(* IEC 61131-3 sources: mocks/test, 17 files *)

(* ---- dummytest.st ---- *)
NAMESPACE dummy
    {Test}
    FUNCTION MyTest
      ; // AxUnit.Assert.Equal(y, x)
    END_FUNCTION
END_NAMESPACE

(* ---- ConfigurableTimerMockTest.st ---- *)
USING System.Timer;
USING AxUnit.Assert;

NAMESPACE Simatic.Ax.Mocks
    /// Example function block that uses multiple OnDelay timers
    FUNCTION_BLOCK MultiTimerFunctionBlock
        VAR_INPUT
            enable1 : BOOL;
            enable2 : BOOL;
            enable3 : BOOL;
        END_VAR
        VAR_OUTPUT
            status1 : STRING;
            status2 : STRING;
            status3 : STRING;
        END_VAR
        VAR
            timer1 : OnDelay;
            timer2 : OnDelay;
            timer3 : OnDelay;
        END_VAR

        // Timer 1: 1 second delay
        timer1(signal := enable1, duration := T#1s);
        IF timer1.output THEN
            status1 := 'T1_ELAPSED';
        ELSE
            status1 := 'T1_WAITING';
        END_IF;

        // Timer 2: 2 second delay
        timer2(signal := enable2, duration := T#2s);
        IF timer2.output THEN
            status2 := 'T2_ELAPSED';
        ELSE
            status2 := 'T2_WAITING';
        END_IF;

        // Timer 3: 5 second delay
        timer3(signal := enable3, duration := T#5s);
        IF timer3.output THEN
            status3 := 'T3_ELAPSED';
        ELSE
            status3 := 'T3_WAITING';
        END_IF;
    END_FUNCTION_BLOCK

    /// Test fixture demonstrating ConfigurableTimerMock usage
    {TestFixture}
    CLASS TestConfigurableTimerMock
        VAR
            testInstance, testInstanceStateless : MultiTimerFunctionBlock;
            payload, payloadStateless : ConfigurableTimerMockPayload;
        END_VAR

        /// Setup method to reset instances before each test
        {TestSetup}
        METHOD PUBLIC TestSetup
            payload := payloadStateless;
            testInstance := testInstanceStateless;
        END_METHOD

        /// Test with Timer 1 elapsed, Timer 2 waiting, Timer 3 elapsed
        /// Timers are identified by call order: 1st call = T1, 2nd call = T2, 3rd call = T3
        {Test}
        METHOD PUBLIC TestMultipleTimersWithDifferentStates
            // Reset counter before test
            payload.ResetCounter();

            // Configure payload: T1=TRUE, T2=FALSE, T3=TRUE (by call order)
            payload.T1_Enabled := TRUE;
            payload.T1_Output := TRUE;
            payload.T1_ElapsedTime := T#1s;

            payload.T2_Enabled := TRUE;
            payload.T2_Output := FALSE;
            payload.T2_ElapsedTime := T#500ms;

            payload.T3_Enabled := TRUE;
            payload.T3_Output := TRUE;
            payload.T3_ElapsedTime := T#5s;

            // Apply mock with payload
            AxUnit.Mocking.Mock(
                mockeeFn := NAME_OF(OnDelay),
                mockFn := NAME_OF(ConfigurableTimerMock),
                payload := payload
            );

            // Execute function block
            // Timer calls happen in order: timer1 (1st call), timer2 (2nd call), timer3 (3rd call)
            testInstance(enable1 := TRUE, enable2 := TRUE, enable3 := TRUE);

            // Verify results
            Equal(expected := 'T1_ELAPSED', actual := testInstance.status1);
            Equal(expected := 'T2_WAITING', actual := testInstance.status2);
            Equal(expected := 'T3_ELAPSED', actual := testInstance.status3);
        END_METHOD

        /// Test with all timers elapsed
        {Test}
        METHOD PUBLIC TestAllTimersElapsed
            // Reset counter before test
            payload.ResetCounter();

            // Configure payload: All timers elapsed
            payload.T1_Enabled := TRUE;
            payload.T1_Output := TRUE;
            payload.T1_ElapsedTime := T#1s;

            payload.T2_Enabled := TRUE;
            payload.T2_Output := TRUE;
            payload.T2_ElapsedTime := T#2s;

            payload.T3_Enabled := TRUE;
            payload.T3_Output := TRUE;
            payload.T3_ElapsedTime := T#5s;

            // Apply mock with payload
            AxUnit.Mocking.Mock(
                mockeeFn := NAME_OF(OnDelay),
                mockFn := NAME_OF(ConfigurableTimerMock),
                payload := payload
            );

            // Execute function block
            testInstance(enable1 := TRUE, enable2 := TRUE, enable3 := TRUE);

            // Verify results
            Equal(expected := 'T1_ELAPSED', actual := testInstance.status1);
            Equal(expected := 'T2_ELAPSED', actual := testInstance.status2);
            Equal(expected := 'T3_ELAPSED', actual := testInstance.status3);
        END_METHOD

        /// Test with only Timer 2 enabled (2nd call)
        {Test}
        METHOD PUBLIC TestOnlyTimer2Enabled
            // Reset counter before test
            payload.ResetCounter();

            // Configure payload: Only T2 enabled and elapsed
            payload.T1_Enabled := FALSE;  // 1st call returns FALSE

            payload.T2_Enabled := TRUE;   // 2nd call returns TRUE
            payload.T2_Output := TRUE;
            payload.T2_ElapsedTime := T#2s;

            payload.T3_Enabled := FALSE;  // 3rd call returns FALSE

            // Apply mock with payload
            AxUnit.Mocking.Mock(
                mockeeFn := NAME_OF(OnDelay),
                mockFn := NAME_OF(ConfigurableTimerMock),
                payload := payload
            );

            // Execute function block
            testInstance(enable1 := TRUE, enable2 := TRUE, enable3 := TRUE);

            // Verify results
            Equal(expected := 'T1_WAITING', actual := testInstance.status1); // 1st call: not enabled
            Equal(expected := 'T2_ELAPSED', actual := testInstance.status2); // 2nd call: enabled and TRUE
            Equal(expected := 'T3_WAITING', actual := testInstance.status3); // 3rd call: not enabled
        END_METHOD
    END_CLASS
END_NAMESPACE

(* ---- ConfigurableTOFMockTest.st ---- *)
USING AxUnit.Assert;

NAMESPACE Simatic.Ax.Mocks
    /// Example function block that uses multiple TOF timers
    FUNCTION_BLOCK MultiTOFFunctionBlock
        VAR_INPUT
            enable1 : BOOL;
            enable2 : BOOL;
            enable3 : BOOL;
        END_VAR
        VAR_OUTPUT
            status1 : STRING;
            status2 : STRING;
            status3 : STRING;
        END_VAR
        VAR
            timer1 : TOF_Mock_true;
            timer2 : TOF_Mock_true;
            timer3 : TOF_Mock_true;
        END_VAR

        // Timer 1: 1 second delay
        timer1(IN := enable1, PT := T#1s);
        IF timer1.Q THEN
            status1 := 'T1_ON';
        ELSE
            status1 := 'T1_OFF';
        END_IF;

        // Timer 2: 2 second delay
        timer2(IN := enable2, PT := T#2s);
        IF timer2.Q THEN
            status2 := 'T2_ON';
        ELSE
            status2 := 'T2_OFF';
        END_IF;

        // Timer 3: 5 second delay
        timer3(IN := enable3, PT := T#5s);
        IF timer3.Q THEN
            status3 := 'T3_ON';
        ELSE
            status3 := 'T3_OFF';
        END_IF;
    END_FUNCTION_BLOCK

    /// Test fixture demonstrating ConfigurableTOFMock usage
    {TestFixture}
    CLASS TestConfigurableTOFMock
        VAR
            testInstance, testInstanceStateless : MultiTOFFunctionBlock;
            payload, payloadStateless : ConfigurableTOFMockPayload;
        END_VAR

        /// Setup method to reset instances before each test
        {TestSetup}
        METHOD PUBLIC TestSetup
            payload := payloadStateless;
            testInstance := testInstanceStateless;
        END_METHOD

        /// Test with Timer 1 ON, Timer 2 OFF, Timer 3 ON
        /// Timers are identified by call order: 1st call = T1, 2nd call = T2, 3rd call = T3
        {Test}
        METHOD PUBLIC TestMultipleTimersWithDifferentStates
            // Reset counter before test
            payload.ResetCounter();

            // Configure payload: T1=TRUE, T2=FALSE, T3=TRUE (by call order)
            payload.T1_Enabled := TRUE;
            payload.T1_Output := TRUE;
            payload.T1_ElapsedTime := T#0ms;

            payload.T2_Enabled := TRUE;
            payload.T2_Output := FALSE;
            payload.T2_ElapsedTime := T#2s;

            payload.T3_Enabled := TRUE;
            payload.T3_Output := TRUE;
            payload.T3_ElapsedTime := T#0ms;

            // Apply mock with payload
            AxUnit.Mocking.Mock(
                mockeeFn := NAME_OF(TOF_Mock_true),
                mockFn := NAME_OF(ConfigurableTOFMock),
                payload := payload
            );

            // Execute function block
            // Timer calls happen in order: timer1 (1st call), timer2 (2nd call), timer3 (3rd call)
            testInstance(enable1 := FALSE, enable2 := FALSE, enable3 := FALSE);

            // Verify results
            Equal(expected := 'T1_ON', actual := testInstance.status1);
            Equal(expected := 'T2_OFF', actual := testInstance.status2);
            Equal(expected := 'T3_ON', actual := testInstance.status3);
        END_METHOD

        /// Test with all timers OFF (delay elapsed)
        {Test}
        METHOD PUBLIC TestAllTimersOff
            // Reset counter before test
            payload.ResetCounter();

            // Configure payload: All timers OFF
            payload.T1_Enabled := TRUE;
            payload.T1_Output := FALSE;
            payload.T1_ElapsedTime := T#1s;

            payload.T2_Enabled := TRUE;
            payload.T2_Output := FALSE;
            payload.T2_ElapsedTime := T#2s;

            payload.T3_Enabled := TRUE;
            payload.T3_Output := FALSE;
            payload.T3_ElapsedTime := T#5s;

            // Apply mock with payload
            AxUnit.Mocking.Mock(
                mockeeFn := NAME_OF(TOF_Mock_true),
                mockFn := NAME_OF(ConfigurableTOFMock),
                payload := payload
            );

            // Execute function block
            testInstance(enable1 := FALSE, enable2 := FALSE, enable3 := FALSE);

            // Verify results
            Equal(expected := 'T1_OFF', actual := testInstance.status1);
            Equal(expected := 'T2_OFF', actual := testInstance.status2);
            Equal(expected := 'T3_OFF', actual := testInstance.status3);
        END_METHOD

        /// Test with only Timer 2 enabled (2nd call)
        {Test}
        METHOD PUBLIC TestOnlyTimer2Enabled
            // Reset counter before test
            payload.ResetCounter();

            // Configure payload: Only T2 enabled and ON
            payload.T1_Enabled := FALSE;  // 1st call returns FALSE

            payload.T2_Enabled := TRUE;   // 2nd call returns TRUE
            payload.T2_Output := TRUE;
            payload.T2_ElapsedTime := T#0ms;

            payload.T3_Enabled := FALSE;  // 3rd call returns FALSE

            // Apply mock with payload
            AxUnit.Mocking.Mock(
                mockeeFn := NAME_OF(TOF_Mock_true),
                mockFn := NAME_OF(ConfigurableTOFMock),
                payload := payload
            );

            // Execute function block
            testInstance(enable1 := FALSE, enable2 := FALSE, enable3 := FALSE);

            // Verify results
            Equal(expected := 'T1_OFF', actual := testInstance.status1); // 1st call: not enabled
            Equal(expected := 'T2_ON', actual := testInstance.status2);  // 2nd call: enabled and TRUE
            Equal(expected := 'T3_OFF', actual := testInstance.status3); // 3rd call: not enabled
        END_METHOD

        /// Test with all timers ON (signal still active or delay not elapsed)
        {Test}
        METHOD PUBLIC TestAllTimersOn
            // Reset counter before test
            payload.ResetCounter();

            // Configure payload: All timers ON
            payload.T1_Enabled := TRUE;
            payload.T1_Output := TRUE;
            payload.T1_ElapsedTime := T#0ms;

            payload.T2_Enabled := TRUE;
            payload.T2_Output := TRUE;
            payload.T2_ElapsedTime := T#0ms;

            payload.T3_Enabled := TRUE;
            payload.T3_Output := TRUE;
            payload.T3_ElapsedTime := T#0ms;

            // Apply mock with payload
            AxUnit.Mocking.Mock(
                mockeeFn := NAME_OF(TOF_Mock_true),
                mockFn := NAME_OF(ConfigurableTOFMock),
                payload := payload
            );

            // Execute function block
            testInstance(enable1 := TRUE, enable2 := TRUE, enable3 := TRUE);

            // Verify results
            Equal(expected := 'T1_ON', actual := testInstance.status1);
            Equal(expected := 'T2_ON', actual := testInstance.status2);
            Equal(expected := 'T3_ON', actual := testInstance.status3);
        END_METHOD
    END_CLASS
END_NAMESPACE

(* ---- ConfigurableTONMockTest.st ---- *)
USING AxUnit.Assert;

NAMESPACE Simatic.Ax.Mocks
    /// Example function block that uses multiple TON timers
    FUNCTION_BLOCK MultiTONFunctionBlock
        VAR_INPUT
            enable1 : BOOL;
            enable2 : BOOL;
            enable3 : BOOL;
        END_VAR
        VAR_OUTPUT
            status1 : STRING;
            status2 : STRING;
            status3 : STRING;
        END_VAR
        VAR
            timer1 : TON_Mock_true;
            timer2 : TON_Mock_true;
            timer3 : TON_Mock_true;
        END_VAR

        // Timer 1: 1 second delay
        timer1(IN := enable1, PT := T#1s);
        IF timer1.Q THEN
            status1 := 'T1_ELAPSED';
        ELSE
            status1 := 'T1_WAITING';
        END_IF;

        // Timer 2: 2 second delay
        timer2(IN := enable2, PT := T#2s);
        IF timer2.Q THEN
            status2 := 'T2_ELAPSED';
        ELSE
            status2 := 'T2_WAITING';
        END_IF;

        // Timer 3: 5 second delay
        timer3(IN := enable3, PT := T#5s);
        IF timer3.Q THEN
            status3 := 'T3_ELAPSED';
        ELSE
            status3 := 'T3_WAITING';
        END_IF;
    END_FUNCTION_BLOCK

    /// Test fixture demonstrating ConfigurableTONMock usage
    {TestFixture}
    CLASS TestConfigurableTONMock
        VAR
            testInstance, testInstanceStateless : MultiTONFunctionBlock;
            payload, payloadStateless : ConfigurableTONMockPayload;
        END_VAR

        /// Setup method to reset instances before each test
        {TestSetup}
        METHOD PUBLIC TestSetup
            payload := payloadStateless;
            testInstance := testInstanceStateless;
        END_METHOD

        /// Test with Timer 1 elapsed, Timer 2 waiting, Timer 3 elapsed
        /// Timers are identified by call order: 1st call = T1, 2nd call = T2, 3rd call = T3
        {Test}
        METHOD PUBLIC TestMultipleTimersWithDifferentStates
            // Reset counter before test
            payload.ResetCounter();

            // Configure payload: T1=TRUE, T2=FALSE, T3=TRUE (by call order)
            payload.T1_Enabled := TRUE;
            payload.T1_Output := TRUE;
            payload.T1_ElapsedTime := T#1s;

            payload.T2_Enabled := TRUE;
            payload.T2_Output := FALSE;
            payload.T2_ElapsedTime := T#500ms;

            payload.T3_Enabled := TRUE;
            payload.T3_Output := TRUE;
            payload.T3_ElapsedTime := T#5s;

            // Apply mock with payload
            AxUnit.Mocking.Mock(
                mockeeFn := NAME_OF(TON_Mock_true),
                mockFn := NAME_OF(ConfigurableTONMock),
                payload := payload
            );

            // Execute function block
            // Timer calls happen in order: timer1 (1st call), timer2 (2nd call), timer3 (3rd call)
            testInstance(enable1 := TRUE, enable2 := TRUE, enable3 := TRUE);

            // Verify results
            Equal(expected := 'T1_ELAPSED', actual := testInstance.status1);
            Equal(expected := 'T2_WAITING', actual := testInstance.status2);
            Equal(expected := 'T3_ELAPSED', actual := testInstance.status3);
        END_METHOD

        /// Test with all timers elapsed
        {Test}
        METHOD PUBLIC TestAllTimersElapsed
            // Reset counter before test
            payload.ResetCounter();

            // Configure payload: All timers elapsed
            payload.T1_Enabled := TRUE;
            payload.T1_Output := TRUE;
            payload.T1_ElapsedTime := T#1s;

            payload.T2_Enabled := TRUE;
            payload.T2_Output := TRUE;
            payload.T2_ElapsedTime := T#2s;

            payload.T3_Enabled := TRUE;
            payload.T3_Output := TRUE;
            payload.T3_ElapsedTime := T#5s;

            // Apply mock with payload
            AxUnit.Mocking.Mock(
                mockeeFn := NAME_OF(TON_Mock_true),
                mockFn := NAME_OF(ConfigurableTONMock),
                payload := payload
            );

            // Execute function block
            testInstance(enable1 := TRUE, enable2 := TRUE, enable3 := TRUE);

            // Verify results
            Equal(expected := 'T1_ELAPSED', actual := testInstance.status1);
            Equal(expected := 'T2_ELAPSED', actual := testInstance.status2);
            Equal(expected := 'T3_ELAPSED', actual := testInstance.status3);
        END_METHOD

        /// Test with only Timer 2 enabled (2nd call)
        {Test}
        METHOD PUBLIC TestOnlyTimer2Enabled
            // Reset counter before test
            payload.ResetCounter();

            // Configure payload: Only T2 enabled and elapsed
            payload.T1_Enabled := FALSE;  // 1st call returns FALSE

            payload.T2_Enabled := TRUE;   // 2nd call returns TRUE
            payload.T2_Output := TRUE;
            payload.T2_ElapsedTime := T#2s;

            payload.T3_Enabled := FALSE;  // 3rd call returns FALSE

            // Apply mock with payload
            AxUnit.Mocking.Mock(
                mockeeFn := NAME_OF(TON_Mock_true),
                mockFn := NAME_OF(ConfigurableTONMock),
                payload := payload
            );

            // Execute function block
            testInstance(enable1 := TRUE, enable2 := TRUE, enable3 := TRUE);

            // Verify results
            Equal(expected := 'T1_WAITING', actual := testInstance.status1); // 1st call: not enabled
            Equal(expected := 'T2_ELAPSED', actual := testInstance.status2); // 2nd call: enabled and TRUE
            Equal(expected := 'T3_WAITING', actual := testInstance.status3); // 3rd call: not enabled
        END_METHOD

        /// Test with all timers waiting
        {Test}
        METHOD PUBLIC TestAllTimersWaiting
            // Reset counter before test
            payload.ResetCounter();

            // Configure payload: All timers waiting
            payload.T1_Enabled := TRUE;
            payload.T1_Output := FALSE;
            payload.T1_ElapsedTime := T#500ms;

            payload.T2_Enabled := TRUE;
            payload.T2_Output := FALSE;
            payload.T2_ElapsedTime := T#1s;

            payload.T3_Enabled := TRUE;
            payload.T3_Output := FALSE;
            payload.T3_ElapsedTime := T#3s;

            // Apply mock with payload
            AxUnit.Mocking.Mock(
                mockeeFn := NAME_OF(TON_Mock_true),
                mockFn := NAME_OF(ConfigurableTONMock),
                payload := payload
            );

            // Execute function block
            testInstance(enable1 := TRUE, enable2 := TRUE, enable3 := TRUE);

            // Verify results
            Equal(expected := 'T1_WAITING', actual := testInstance.status1);
            Equal(expected := 'T2_WAITING', actual := testInstance.status2);
            Equal(expected := 'T3_WAITING', actual := testInstance.status3);
        END_METHOD
    END_CLASS
END_NAMESPACE

(* ---- ExampleMockTimer.st ---- *)
USING System.Timer;
USING AxUnit.Assert;

NAMESPACE Simatic.Ax.Mocks
    FUNCTION_BLOCK FunctionBlockWhichUsesTimer
        VAR_INPUT
            enable : BOOL;
        END_VAR
        VAR_OUTPUT
            timerStatus : STRING;
        END_VAR

        VAR
            ton : OnDelay;
        END_VAR

        ton(signal := enable, duration := T#10s);

        IF (ton.output) THEN
            timerStatus := 'ELAPSED';
        ELSIF (ton.signal AND NOT ton.output) THEN
            timerStatus := 'RUNNING';
        ELSIF (NOT ton.signal) THEN
            timerStatus := 'IDLE';
        END_IF;
        ;
    END_FUNCTION_BLOCK

    {TestFixture}
    CLASS TestFunctionBlockWhichUsesTimer
        VAR
            testInstance : FunctionBlockWhichUsesTimer;
        END_VAR

        {Test}
        METHOD PUBLIC FunctionBlockReturnsIdleWhenNotEnabled
            testInstance(enable := FALSE);
            Equal(expected := 'ELAPSED', actual := testInstance.timerStatus);
        END_METHOD

        {Test}
        METHOD PUBLIC FunctionBlockReturnsRunningWhenEnabledAndTimeIsNotElapsed
            testInstance(enable := TRUE);
            Equal(expected := 'RUNNING', actual := testInstance.timerStatus);
        END_METHOD

        {Test}
        METHOD PUBLIC FunctionBlockReturnsElapsedWhenEnabledAndTimeHasElapsed
            testInstance(enable := TRUE);
            Equal(expected := 'ELAPSED', actual := testInstance.timerStatus);
        END_METHOD
    END_CLASS
END_NAMESPACE

(* ---- FooFB_ConfigurableMock_Test.st ---- *)
USING AxUnit.Assert;
USING System.Timer;

NAMESPACE Simatic.Ax.Mocks
    /// Test fixture for FbWithThreeTimers using ConfigurableTimerMock
    /// This demonstrates call-order based timer mocking
    /// Uses stateless pattern to ensure test isolation
    {TestFixture}
    CLASS TestFbWithThreeTimers_ConfigurableMock
        VAR
            myFB, myFBStateless : FbWithThreeTimers;
            payload, payloadStateless : ConfigurableTimerMockPayload;
        END_VAR

        /// Setup method to reset instances before each test
        {TestSetup}
        METHOD PUBLIC TestSetup
            payload := payloadStateless;
            myFB := myFBStateless;
        END_METHOD

        /// Test scenario: T1 elapsed, T2 waiting, T3 elapsed
        {Test}
        METHOD PUBLIC Test_T1_Elapsed_T2_Waiting_T3_Elapsed
            // Reset counter before test
            payload.ResetCounter();

            // Configure timers by call order
            // T1 is 1st call - elapsed
            payload.T1_Enabled := TRUE;
            payload.T1_Output := TRUE;
            payload.T1_ElapsedTime := T#10s;

            // T2 is 2nd call - waiting
            payload.T2_Enabled := TRUE;
            payload.T2_Output := FALSE;
            payload.T2_ElapsedTime := T#5s;

            // T3 is 3rd call - elapsed
            payload.T3_Enabled := TRUE;
            payload.T3_Output := TRUE;
            payload.T3_ElapsedTime := T#30s;

            // Apply mock
            AxUnit.Mocking.Mock(
                mockeeFn := NAME_OF(OnDelay),
                mockFn := NAME_OF(ConfigurableTimerMock),
                payload := payload
            );

            // Execute function block
            myFB.SignalT1 := TRUE;
            myFB.SignalT2 := TRUE;
            myFB.SignalT3 := TRUE;
            myFB();

            // Verify results
            Equal(expected := TRUE, actual := myFB.OutputT1);
            Equal(expected := FALSE, actual := myFB.OutputT2);
            Equal(expected := TRUE, actual := myFB.OutputT3);
        END_METHOD

        /// Test scenario: All timers elapsed
        {Test}
        METHOD PUBLIC Test_AllTimersElapsed
            payload.ResetCounter();

            // All timers elapsed
            payload.T1_Enabled := TRUE;
            payload.T1_Output := TRUE;
            payload.T1_ElapsedTime := T#10s;

            payload.T2_Enabled := TRUE;
            payload.T2_Output := TRUE;
            payload.T2_ElapsedTime := T#20s;

            payload.T3_Enabled := TRUE;
            payload.T3_Output := TRUE;
            payload.T3_ElapsedTime := T#30s;

            // Apply mock
            AxUnit.Mocking.Mock(
                mockeeFn := NAME_OF(OnDelay),
                mockFn := NAME_OF(ConfigurableTimerMock),
                payload := payload
            );

            // Execute
            myFB.SignalT1 := TRUE;
            myFB.SignalT2 := TRUE;
            myFB.SignalT3 := TRUE;
            myFB();

            // Verify all outputs are TRUE
            Equal(expected := TRUE, actual := myFB.OutputT1);
            Equal(expected := TRUE, actual := myFB.OutputT2);
            Equal(expected := TRUE, actual := myFB.OutputT3);
        END_METHOD

        /// Test scenario: All timers waiting
        {Test}
        METHOD PUBLIC Test_AllTimersWaiting
            payload.ResetCounter();

            // All timers waiting
            payload.T1_Enabled := TRUE;
            payload.T1_Output := FALSE;
            payload.T1_ElapsedTime := T#3s;

            payload.T2_Enabled := TRUE;
            payload.T2_Output := FALSE;
            payload.T2_ElapsedTime := T#7s;

            payload.T3_Enabled := TRUE;
            payload.T3_Output := FALSE;
            payload.T3_ElapsedTime := T#15s;

            // Apply mock
            AxUnit.Mocking.Mock(
                mockeeFn := NAME_OF(OnDelay),
                mockFn := NAME_OF(ConfigurableTimerMock),
                payload := payload
            );

            // Execute
            myFB.SignalT1 := TRUE;
            myFB.SignalT2 := TRUE;
            myFB.SignalT3 := TRUE;
            myFB();

            // Verify all outputs are FALSE
            Equal(expected := FALSE, actual := myFB.OutputT1);
            Equal(expected := FALSE, actual := myFB.OutputT2);
            Equal(expected := FALSE, actual := myFB.OutputT3);
        END_METHOD

        /// Test scenario: Only T2 enabled (others disabled)
        {Test}
        METHOD PUBLIC Test_OnlyT2Enabled
            payload.ResetCounter();

            // Only T2 enabled at position 2
            payload.T1_Enabled := FALSE;  // 1st call - not configured

            payload.T2_Enabled := TRUE;   // 2nd call - configured
            payload.T2_Output := TRUE;
            payload.T2_ElapsedTime := T#20s;

            payload.T3_Enabled := FALSE;  // 3rd call - not configured

            // Apply mock
            AxUnit.Mocking.Mock(
                mockeeFn := NAME_OF(OnDelay),
                mockFn := NAME_OF(ConfigurableTimerMock),
                payload := payload
            );

            // Execute
            myFB.SignalT1 := TRUE;
            myFB.SignalT2 := TRUE;
            myFB.SignalT3 := TRUE;
            myFB();

            // Verify: T1 and T3 default to FALSE, T2 is TRUE
            Equal(expected := FALSE, actual := myFB.OutputT1);
            Equal(expected := TRUE, actual := myFB.OutputT2);
            Equal(expected := FALSE, actual := myFB.OutputT3);
        END_METHOD

        /// Test scenario: Mixed signals - some enabled, some disabled
        {Test}
        METHOD PUBLIC Test_MixedSignals
            payload.ResetCounter();

            // Configure all timers as elapsed
            payload.T1_Enabled := TRUE;
            payload.T1_Output := TRUE;
            payload.T1_ElapsedTime := T#10s;

            payload.T2_Enabled := TRUE;
            payload.T2_Output := TRUE;
            payload.T2_ElapsedTime := T#20s;

            payload.T3_Enabled := TRUE;
            payload.T3_Output := TRUE;
            payload.T3_ElapsedTime := T#30s;

            // Apply mock
            AxUnit.Mocking.Mock(
                mockeeFn := NAME_OF(OnDelay),
                mockFn := NAME_OF(ConfigurableTimerMock),
                payload := payload
            );

            // Execute with mixed signals
            myFB.SignalT1 := TRUE;   // Enabled
            myFB.SignalT2 := FALSE;  // Disabled
            myFB.SignalT3 := TRUE;   // Enabled
            myFB();

            // Verify: Mock returns configured values regardless of signal
            // (This is the mock behavior - it ignores the signal input)
            Equal(expected := TRUE, actual := myFB.OutputT1);
            Equal(expected := TRUE, actual := myFB.OutputT2);
            Equal(expected := TRUE, actual := myFB.OutputT3);
        END_METHOD
    END_CLASS
END_NAMESPACE

(* ---- FooFB_IdentifierMock_Test.st ---- *)
USING AxUnit.Assert;
USING System.Timer;

NAMESPACE Simatic.Ax.Mocks
    /// Test fixture for FbWithThreeTimers using IdentifierBasedTimerMock
    /// This demonstrates position-based timer mocking with explicit call positions
    /// Uses stateless pattern to ensure test isolation
    {TestFixture}
    CLASS TestFbWithThreeTimers_IdentifierMock
        VAR
            myFB, myFBStateless : FbWithThreeTimers;
            payload, payloadStateless : IdentifierBasedOnDelayMockPayload;
        END_VAR

        /// Setup method to reset instances before each test
        {TestSetup}
        METHOD PUBLIC TestSetup
            payload := payloadStateless;
            myFB := myFBStateless;
        END_METHOD

        /// Test scenario: T1 elapsed, T2 waiting, T3 elapsed
        /// Using explicit call positions
        {Test}
        METHOD PUBLIC Test_T1_Elapsed_T2_Waiting_T3_Elapsed
            // Reset counter before test
            payload.ResetCounter();

            // Configure timers by explicit call position
            // T1 at position 1 - elapsed
            payload.T1_Enabled := TRUE;
            payload.T1_CallPosition := 1;  // 1st call
            payload.T1_Output := TRUE;
            payload.T1_ElapsedTime := T#10s;

            // T2 at position 2 - waiting
            payload.T2_Enabled := TRUE;
            payload.T2_CallPosition := 2;  // 2nd call
            payload.T2_Output := FALSE;
            payload.T2_ElapsedTime := T#5s;

            // T3 at position 3 - elapsed
            payload.T3_Enabled := TRUE;
            payload.T3_CallPosition := 3;  // 3rd call
            payload.T3_Output := TRUE;
            payload.T3_ElapsedTime := T#30s;

            // Apply mock
            AxUnit.Mocking.Mock(
                mockeeFn := NAME_OF(OnDelay),
                mockFn := NAME_OF(IdentifierBasedOnDelayMock),
                payload := payload
            );

            // Execute function block
            myFB.SignalT1 := TRUE;
            myFB.SignalT2 := TRUE;
            myFB.SignalT3 := TRUE;
            myFB();

            // Verify results
            Equal(expected := TRUE, actual := myFB.OutputT1);
            Equal(expected := FALSE, actual := myFB.OutputT2);
            Equal(expected := TRUE, actual := myFB.OutputT3);
        END_METHOD

        /// Test scenario: All timers elapsed
        {Test}
        METHOD PUBLIC Test_AllTimersElapsed
            payload.ResetCounter();

            // All timers elapsed at their respective positions
            payload.T1_Enabled := TRUE;
            payload.T1_CallPosition := 1;
            payload.T1_Output := TRUE;
            payload.T1_ElapsedTime := T#10s;

            payload.T2_Enabled := TRUE;
            payload.T2_CallPosition := 2;
            payload.T2_Output := TRUE;
            payload.T2_ElapsedTime := T#20s;

            payload.T3_Enabled := TRUE;
            payload.T3_CallPosition := 3;
            payload.T3_Output := TRUE;
            payload.T3_ElapsedTime := T#30s;

            // Apply mock
            AxUnit.Mocking.Mock(
                mockeeFn := NAME_OF(OnDelay),
                mockFn := NAME_OF(IdentifierBasedOnDelayMock),
                payload := payload
            );

            // Execute
            myFB.SignalT1 := TRUE;
            myFB.SignalT2 := TRUE;
            myFB.SignalT3 := TRUE;
            myFB();

            // Verify all outputs are TRUE
            Equal(expected := TRUE, actual := myFB.OutputT1);
            Equal(expected := TRUE, actual := myFB.OutputT2);
            Equal(expected := TRUE, actual := myFB.OutputT3);
        END_METHOD

        /// Test scenario: All timers waiting
        {Test}
        METHOD PUBLIC Test_AllTimersWaiting
            payload.ResetCounter();

            // All timers waiting
            payload.T1_Enabled := TRUE;
            payload.T1_CallPosition := 1;
            payload.T1_Output := FALSE;
            payload.T1_ElapsedTime := T#3s;

            payload.T2_Enabled := TRUE;
            payload.T2_CallPosition := 2;
            payload.T2_Output := FALSE;
            payload.T2_ElapsedTime := T#7s;

            payload.T3_Enabled := TRUE;
            payload.T3_CallPosition := 3;
            payload.T3_Output := FALSE;
            payload.T3_ElapsedTime := T#15s;

            // Apply mock
            AxUnit.Mocking.Mock(
                mockeeFn := NAME_OF(OnDelay),
                mockFn := NAME_OF(IdentifierBasedOnDelayMock),
                payload := payload
            );

            // Execute
            myFB.SignalT1 := TRUE;
            myFB.SignalT2 := TRUE;
            myFB.SignalT3 := TRUE;
            myFB();

            // Verify all outputs are FALSE
            Equal(expected := FALSE, actual := myFB.OutputT1);
            Equal(expected := FALSE, actual := myFB.OutputT2);
            Equal(expected := FALSE, actual := myFB.OutputT3);
        END_METHOD

        /// Test scenario: Only T2 configured at position 2
        {Test}
        METHOD PUBLIC Test_OnlyT2Configured
            payload.ResetCounter();

            // Only configure T2 at position 2
            payload.T1_Enabled := FALSE;  // Position 1 - not configured

            payload.T2_Enabled := TRUE;   // Position 2 - configured
            payload.T2_CallPosition := 2;
            payload.T2_Output := TRUE;
            payload.T2_ElapsedTime := T#20s;

            payload.T3_Enabled := FALSE;  // Position 3 - not configured

            // Apply mock
            AxUnit.Mocking.Mock(
                mockeeFn := NAME_OF(OnDelay),
                mockFn := NAME_OF(IdentifierBasedOnDelayMock),
                payload := payload
            );

            // Execute
            myFB.SignalT1 := TRUE;
            myFB.SignalT2 := TRUE;
            myFB.SignalT3 := TRUE;
            myFB();

            // Verify: T1 and T3 default to FALSE, T2 is TRUE
            Equal(expected := FALSE, actual := myFB.OutputT1);
            Equal(expected := TRUE, actual := myFB.OutputT2);
            Equal(expected := FALSE, actual := myFB.OutputT3);
        END_METHOD

        /// Test scenario: Non-sequential positions (demonstrating flexibility)
        /// Configure T1 at position 3, T3 at position 1 (swapped)
        {Test}
        METHOD PUBLIC Test_NonSequentialPositions
            payload.ResetCounter();

            // Swap positions: T3 at position 1, T1 at position 3
            payload.T1_Enabled := TRUE;
            payload.T1_CallPosition := 3;  // T1 configured for 3rd call
            payload.T1_Output := TRUE;
            payload.T1_ElapsedTime := T#10s;

            payload.T2_Enabled := TRUE;
            payload.T2_CallPosition := 2;  // T2 at 2nd call (normal)
            payload.T2_Output := FALSE;
            payload.T2_ElapsedTime := T#5s;

            payload.T3_Enabled := TRUE;
            payload.T3_CallPosition := 1;  // T3 configured for 1st call
            payload.T3_Output := TRUE;
            payload.T3_ElapsedTime := T#30s;

            // Apply mock
            AxUnit.Mocking.Mock(
                mockeeFn := NAME_OF(OnDelay),
                mockFn := NAME_OF(IdentifierBasedOnDelayMock),
                payload := payload
            );

            // Execute
            myFB.SignalT1 := TRUE;
            myFB.SignalT2 := TRUE;
            myFB.SignalT3 := TRUE;
            myFB();

            // Verify:
            // 1st call (T1 in code) gets T3 config -> TRUE
            // 2nd call (T2 in code) gets T2 config -> FALSE
            // 3rd call (T3 in code) gets T1 config -> TRUE
            Equal(expected := TRUE, actual := myFB.OutputT1);   // Gets T3 config
            Equal(expected := FALSE, actual := myFB.OutputT2);  // Gets T2 config
            Equal(expected := TRUE, actual := myFB.OutputT3);   // Gets T1 config
        END_METHOD

        /// Test scenario: Partial elapsed times
        /// Demonstrates setting specific elapsed times for each timer
        {Test}
        METHOD PUBLIC Test_PartialElapsedTimes
            payload.ResetCounter();

            // Configure with specific elapsed times
            payload.T1_Enabled := TRUE;
            payload.T1_CallPosition := 1;
            payload.T1_Output := FALSE;  // Not elapsed yet
            payload.T1_ElapsedTime := T#7s;  // 7 of 10 seconds

            payload.T2_Enabled := TRUE;
            payload.T2_CallPosition := 2;
            payload.T2_Output := FALSE;  // Not elapsed yet
            payload.T2_ElapsedTime := T#15s;  // 15 of 20 seconds

            payload.T3_Enabled := TRUE;
            payload.T3_CallPosition := 3;
            payload.T3_Output := TRUE;  // Elapsed
            payload.T3_ElapsedTime := T#30s;  // Full 30 seconds

            // Apply mock
            AxUnit.Mocking.Mock(
                mockeeFn := NAME_OF(OnDelay),
                mockFn := NAME_OF(IdentifierBasedOnDelayMock),
                payload := payload
            );

            // Execute
            myFB.SignalT1 := TRUE;
            myFB.SignalT2 := TRUE;
            myFB.SignalT3 := TRUE;
            myFB();

            // Verify outputs
            Equal(expected := FALSE, actual := myFB.OutputT1);  // 7s < 10s
            Equal(expected := FALSE, actual := myFB.OutputT2);  // 15s < 20s
            Equal(expected := TRUE, actual := myFB.OutputT3);   // 30s = 30s
        END_METHOD
    END_CLASS
END_NAMESPACE

(* ---- FooFbWithThreeTimers.st ---- *)
USING AxUnit.Assert;
USING System.Timer;
NAMESPACE Simatic.Ax.Mocks

    FUNCTION_BLOCK FbWithThreeTimers
        VAR_INPUT
            SignalT1 : BOOL;
            SignalT2 : BOOL;
            SignalT3 : BOOL;
        END_VAR
        VAR_OUTPUT
            OutputT1 : BOOL;
            OutputT2 : BOOL;
            OutputT3 : BOOL;
        END_VAR
        VAR
            T1 : OnDelay;
            T2 : OnDelay;
            T3 : OnDelay;
        END_VAR
        T1(Signal := SignalT1, Duration := LTIME#10S, Output => OutputT1);
        T2(Signal := SignalT2, Duration := LTIME#20S, Output => OutputT2);
        T3(Signal := SignalT3, Duration := LTIME#30S, Output => OutputT3);
    END_FUNCTION_BLOCK
END_NAMESPACE

(* ---- IdentifierBasedOffDelayMockTest.st ---- *)
USING System.Timer;
USING AxUnit.Assert;

NAMESPACE Simatic.Ax.Mocks
    /// Example function block with conditional OffDelay timer usage
    FUNCTION_BLOCK ConditionalOffDelayFunctionBlock
        VAR_INPUT
            mode : INT;  // 1, 2, or 3 to select which timer to use
        END_VAR
        VAR_OUTPUT
            result : STRING;
        END_VAR
        VAR
            timer1 : OffDelay;
            timer2 : OffDelay;
            timer3 : OffDelay;
        END_VAR

        // Conditional timer usage based on mode
        IF mode = 1 THEN
            timer1(signal := FALSE, duration := T#1s);
            IF timer1.output THEN
                result := 'MODE1_ON';
            ELSE
                result := 'MODE1_OFF';
            END_IF;
        ELSIF mode = 2 THEN
            timer2(signal := FALSE, duration := T#2s);
            IF timer2.output THEN
                result := 'MODE2_ON';
            ELSE
                result := 'MODE2_OFF';
            END_IF;
        ELSIF mode = 3 THEN
            timer3(signal := FALSE, duration := T#5s);
            IF timer3.output THEN
                result := 'MODE3_ON';
            ELSE
                result := 'MODE3_OFF';
            END_IF;
        ELSE
            result := 'INVALID_MODE';
        END_IF;
    END_FUNCTION_BLOCK

    /// Test fixture demonstrating IdentifierBasedOffDelayMock usage
    {TestFixture}
    CLASS TestIdentifierBasedOffDelayMock
        VAR
            testInstance, testInstanceStateless : ConditionalOffDelayFunctionBlock;
            payload, payloadStateless : IdentifierBasedOffDelayMockPayload;
        END_VAR

        /// Setup method to reset instances before each test
        {TestSetup}
        METHOD PUBLIC TestSetup
            payload := payloadStateless;
            testInstance := testInstanceStateless;
        END_METHOD

        /// Test Mode 1 - Timer at position 1 should be ON
        {Test}
        METHOD PUBLIC TestMode1TimerOn
            // Reset counter before test
            payload.ResetCounter();

            // Configure Timer 1 (1st call position) to be ON
            payload.T1_Enabled := TRUE;
            payload.T1_CallPosition := 1;
            payload.T1_Output := TRUE;
            payload.T1_ElapsedTime := T#0ms;

            // Apply mock with payload
            AxUnit.Mocking.Mock(
                mockeeFn := NAME_OF(OffDelay),
                mockFn := NAME_OF(IdentifierBasedOffDelayMock),
                payload := payload
            );

            // Execute function block in mode 1
            testInstance(mode := 1);

            // Verify result
            Equal(expected := 'MODE1_ON', actual := testInstance.result);
        END_METHOD

        /// Test Mode 2 - Timer at position 1 should be OFF
        {Test}
        METHOD PUBLIC TestMode2TimerOff
            // Reset counter before test
            payload.ResetCounter();

            // Configure Timer 1 (1st call position) to be OFF
            payload.T1_Enabled := TRUE;
            payload.T1_CallPosition := 1;
            payload.T1_Output := FALSE;
            payload.T1_ElapsedTime := T#2s;

            // Apply mock with payload
            AxUnit.Mocking.Mock(
                mockeeFn := NAME_OF(OffDelay),
                mockFn := NAME_OF(IdentifierBasedOffDelayMock),
                payload := payload
            );

            // Execute function block in mode 2
            testInstance(mode := 2);

            // Verify result
            Equal(expected := 'MODE2_OFF', actual := testInstance.result);
        END_METHOD

        /// Test Mode 3 - Timer at position 1 should be ON
        {Test}
        METHOD PUBLIC TestMode3TimerOn
            // Reset counter before test
            payload.ResetCounter();

            // Configure Timer 1 (1st call position) to be ON
            payload.T1_Enabled := TRUE;
            payload.T1_CallPosition := 1;
            payload.T1_Output := TRUE;
            payload.T1_ElapsedTime := T#0ms;

            // Apply mock with payload
            AxUnit.Mocking.Mock(
                mockeeFn := NAME_OF(OffDelay),
                mockFn := NAME_OF(IdentifierBasedOffDelayMock),
                payload := payload
            );

            // Execute function block in mode 3
            testInstance(mode := 3);

            // Verify result
            Equal(expected := 'MODE3_ON', actual := testInstance.result);
        END_METHOD

        /// Test with multiple configured timers - only matching position is used
        {Test}
        METHOD PUBLIC TestMultipleConfiguredTimers
            // Reset counter before test
            payload.ResetCounter();

            // Configure multiple timers with different call positions
            payload.T1_Enabled := TRUE;
            payload.T1_CallPosition := 1;
            payload.T1_Output := FALSE;
            payload.T1_ElapsedTime := T#1s;

            payload.T2_Enabled := TRUE;
            payload.T2_CallPosition := 2;
            payload.T2_Output := TRUE;
            payload.T2_ElapsedTime := T#0ms;

            // Apply mock with payload
            AxUnit.Mocking.Mock(
                mockeeFn := NAME_OF(OffDelay),
                mockFn := NAME_OF(IdentifierBasedOffDelayMock),
                payload := payload
            );

            // Execute function block in mode 2 (should match T2 at position 1, but T1 is at position 1)
            // Since mode 2 calls timer2, it's the 1st call, so T1 matches
            testInstance(mode := 2);

            // Verify result - T1 configuration is used (position 1, OFF)
            Equal(expected := 'MODE2_OFF', actual := testInstance.result);
        END_METHOD
    END_CLASS
END_NAMESPACE

(* ---- IdentifierBasedTimerMockTest.st ---- *)
USING System.Timer;
USING AxUnit.Assert;

NAMESPACE Simatic.Ax.Mocks
    /// Example function block with conditional timer usage
    /// Depending on mode, different timers are called at different positions
    FUNCTION_BLOCK ConditionalTimerExample
        VAR_INPUT
            mode : INT;         // 1 = use T1+T2, 2 = use T1+T3
            enable : BOOL;
        END_VAR
        VAR_OUTPUT
            status : STRING;
        END_VAR
        VAR
            timer1 : OnDelay;   // Always used at position 1
            timer2 : OnDelay;   // Used at position 2 in mode 1
            timer3 : OnDelay;   // Used at position 2 in mode 2
        END_VAR

        // Timer 1 is always called first (position 1)
        timer1(signal := enable, duration := T#1s);

        IF mode = 1 THEN
            // Mode 1: Timer 2 is called at position 2
            timer2(signal := enable, duration := T#2s);

            IF timer1.output AND timer2.output THEN
                status := 'MODE1_BOTH_ELAPSED';
            ELSIF timer1.output THEN
                status := 'MODE1_T1_ELAPSED';
            ELSE
                status := 'MODE1_WAITING';
            END_IF;

        ELSIF mode = 2 THEN
            // Mode 2: Timer 3 is called at position 2
            timer3(signal := enable, duration := T#3s);

            IF timer1.output AND timer3.output THEN
                status := 'MODE2_BOTH_ELAPSED';
            ELSIF timer1.output THEN
                status := 'MODE2_T1_ELAPSED';
            ELSE
                status := 'MODE2_WAITING';
            END_IF;
        END_IF;
    END_FUNCTION_BLOCK

    /// Test fixture demonstrating IdentifierBasedTimerMock with conditional timers
    {TestFixture}
    CLASS TestIdentifierBasedTimerMock
        VAR
            testInstance, testInstanceStateless : ConditionalTimerExample;
            testInstanceMulti, testInstanceMultiStateless : MultiTimerFunctionBlock;
            payload, payloadStateless : IdentifierBasedTimerMockPayload;
        END_VAR

        {TestSetup}
        METHOD PUBLIC TestSetup
            payload := payloadStateless;
            testInstance := testInstanceStateless;
            testInstanceMulti := testInstanceMultiStateless;
        END_METHOD

        /// Test Mode 1: T1 at position 1, T2 at position 2
        {Test}
        METHOD PUBLIC TestMode1_BothTimersElapsed
            payload.ResetCounter();

            // Timer 1: Position 1 (always first call)
            payload.T1_Enabled := TRUE;
            payload.T1_CallPosition := 1;  // 1st call
            payload.T1_Output := TRUE;
            payload.T1_ElapsedTime := T#1s;

            // Timer 2: Position 2 (second call in mode 1)
            payload.T2_Enabled := TRUE;
            payload.T2_CallPosition := 2;  // 2nd call
            payload.T2_Output := TRUE;
            payload.T2_ElapsedTime := T#2s;

            // Timer 3: not called in mode 1
            payload.T3_Enabled := FALSE;

            // Apply mock
            AxUnit.Mocking.Mock(
                mockeeFn := NAME_OF(OnDelay),
                mockFn := NAME_OF(IdentifierBasedTimerMock),
                payload := payload
            );

            // Execute in mode 1
            testInstance(mode := 1, enable := TRUE);

            // Verify both timers elapsed
            Equal(expected := 'MODE1_BOTH_ELAPSED', actual := testInstance.status);
        END_METHOD

        /// Test Mode 1: T1 elapsed, T2 waiting
        {Test}
        METHOD PUBLIC TestMode1_OnlyT1Elapsed
            payload.ResetCounter();

            // Timer 1: Position 1, elapsed
            payload.T1_Enabled := TRUE;
            payload.T1_CallPosition := 1;
            payload.T1_Output := TRUE;
            payload.T1_ElapsedTime := T#1s;

            // Timer 2: Position 2, not elapsed
            payload.T2_Enabled := TRUE;
            payload.T2_CallPosition := 2;
            payload.T2_Output := FALSE;
            payload.T2_ElapsedTime := T#500ms;

            // Timer 3: not called in mode 1
            payload.T3_Enabled := FALSE;

            // Apply mock
            AxUnit.Mocking.Mock(
                mockeeFn := NAME_OF(OnDelay),
                mockFn := NAME_OF(IdentifierBasedTimerMock),
                payload := payload
            );

            // Execute in mode 1
            testInstance(mode := 1, enable := TRUE);

            // Verify only T1 elapsed
            Equal(expected := 'MODE1_T1_ELAPSED', actual := testInstance.status);
        END_METHOD

        /// Test Mode 2: T1 at position 1, T3 at position 2
        {Test}
        METHOD PUBLIC TestMode2_BothTimersElapsed
            payload.ResetCounter();

            // Timer 1: Position 1 (always first call)
            payload.T1_Enabled := TRUE;
            payload.T1_CallPosition := 1;  // 1st call
            payload.T1_Output := TRUE;
            payload.T1_ElapsedTime := T#1s;

            // Timer 2: not called in mode 2
            payload.T2_Enabled := FALSE;

            // Timer 3: Position 2 (second call in mode 2)
            payload.T3_Enabled := TRUE;
            payload.T3_CallPosition := 2;  // 2nd call
            payload.T3_Output := TRUE;
            payload.T3_ElapsedTime := T#3s;

            // Apply mock
            AxUnit.Mocking.Mock(
                mockeeFn := NAME_OF(OnDelay),
                mockFn := NAME_OF(IdentifierBasedTimerMock),
                payload := payload
            );

            // Execute in mode 2
            testInstance(mode := 2, enable := TRUE);

            // Verify both timers elapsed
            Equal(expected := 'MODE2_BOTH_ELAPSED', actual := testInstance.status);
        END_METHOD

        /// Test Mode 2: T1 elapsed, T3 waiting
        {Test}
        METHOD PUBLIC TestMode2_OnlyT1Elapsed
            payload.ResetCounter();

            // Timer 1: Position 1, elapsed
            payload.T1_Enabled := TRUE;
            payload.T1_CallPosition := 1;
            payload.T1_Output := TRUE;
            payload.T1_ElapsedTime := T#1s;

            // Timer 2: not called in mode 2
            payload.T2_Enabled := FALSE;

            // Timer 3: Position 2, not elapsed
            payload.T3_Enabled := TRUE;
            payload.T3_CallPosition := 2;
            payload.T3_Output := FALSE;
            payload.T3_ElapsedTime := T#1500ms;

            // Apply mock
            AxUnit.Mocking.Mock(
                mockeeFn := NAME_OF(OnDelay),
                mockFn := NAME_OF(IdentifierBasedTimerMock),
                payload := payload
            );

            // Execute in mode 2
            testInstance(mode := 2, enable := TRUE);

            // Verify only T1 elapsed
            Equal(expected := 'MODE2_T1_ELAPSED', actual := testInstance.status);
        END_METHOD

        /// Test with 3 sequential timers (no conditional logic)
        {Test}
        METHOD PUBLIC TestSequentialTimers
            payload.ResetCounter();

            // Configure 3 timers at positions 1, 2, 3
            payload.T1_Enabled := TRUE;
            payload.T1_CallPosition := 1;
            payload.T1_Output := TRUE;
            payload.T1_ElapsedTime := T#1s;

            payload.T2_Enabled := TRUE;
            payload.T2_CallPosition := 2;
            payload.T2_Output := FALSE;
            payload.T2_ElapsedTime := T#500ms;

            payload.T3_Enabled := TRUE;
            payload.T3_CallPosition := 3;
            payload.T3_Output := TRUE;
            payload.T3_ElapsedTime := T#5s;

            // Apply mock
            AxUnit.Mocking.Mock(
                mockeeFn := NAME_OF(OnDelay),
                mockFn := NAME_OF(IdentifierBasedTimerMock),
                payload := payload
            );

            // Execute
            testInstanceMulti(enable1 := TRUE, enable2 := TRUE, enable3 := TRUE);

            // Verify results
            Equal(expected := 'T1_ELAPSED', actual := testInstanceMulti.status1);
            Equal(expected := 'T2_WAITING', actual := testInstanceMulti.status2);
            Equal(expected := 'T3_ELAPSED', actual := testInstanceMulti.status3);
        END_METHOD
    END_CLASS
END_NAMESPACE

(* ---- IdentifierBasedTOFMockTest.st ---- *)
USING AxUnit.Assert;

NAMESPACE Simatic.Ax.Mocks
    /// Example function block with conditional TOF timer usage
    FUNCTION_BLOCK ConditionalTOFFunctionBlock
        VAR_INPUT
            mode : INT;  // 1, 2, or 3 to select which timer to use
        END_VAR
        VAR_OUTPUT
            result : STRING;
        END_VAR
        VAR
            timer1 : TOF_Mock_true;
            timer2 : TOF_Mock_true;
            timer3 : TOF_Mock_true;
        END_VAR

        // Conditional timer usage based on mode
        IF mode = 1 THEN
            timer1(IN := FALSE, PT := T#1s);
            IF timer1.Q THEN
                result := 'MODE1_ON';
            ELSE
                result := 'MODE1_OFF';
            END_IF;
        ELSIF mode = 2 THEN
            timer2(IN := FALSE, PT := T#2s);
            IF timer2.Q THEN
                result := 'MODE2_ON';
            ELSE
                result := 'MODE2_OFF';
            END_IF;
        ELSIF mode = 3 THEN
            timer3(IN := FALSE, PT := T#5s);
            IF timer3.Q THEN
                result := 'MODE3_ON';
            ELSE
                result := 'MODE3_OFF';
            END_IF;
        ELSE
            result := 'INVALID_MODE';
        END_IF;
    END_FUNCTION_BLOCK

    /// Test fixture demonstrating IdentifierBasedTOFMock usage
    {TestFixture}
    CLASS TestIdentifierBasedTOFMock
        VAR
            testInstance, testInstanceStateless : ConditionalTOFFunctionBlock;
            payload, payloadStateless : IdentifierBasedTOFMockPayload;
        END_VAR

        /// Setup method to reset instances before each test
        {TestSetup}
        METHOD PUBLIC TestSetup
            payload := payloadStateless;
            testInstance := testInstanceStateless;
        END_METHOD

        /// Test Mode 1 - Timer at position 1 should be ON
        {Test}
        METHOD PUBLIC TestMode1TimerOn
            // Reset counter before test
            payload.ResetCounter();

            // Configure Timer 1 (1st call position) to be ON
            payload.T1_Enabled := TRUE;
            payload.T1_CallPosition := 1;
            payload.T1_Output := TRUE;
            payload.T1_ElapsedTime := T#0ms;

            // Apply mock with payload
            AxUnit.Mocking.Mock(
                mockeeFn := NAME_OF(TOF_Mock_true),
                mockFn := NAME_OF(IdentifierBasedTOFMock),
                payload := payload
            );

            // Execute function block in mode 1
            testInstance(mode := 1);

            // Verify result
            Equal(expected := 'MODE1_ON', actual := testInstance.result);
        END_METHOD

        /// Test Mode 2 - Timer at position 1 should be OFF
        {Test}
        METHOD PUBLIC TestMode2TimerOff
            // Reset counter before test
            payload.ResetCounter();

            // Configure Timer 1 (1st call position) to be OFF
            payload.T1_Enabled := TRUE;
            payload.T1_CallPosition := 1;
            payload.T1_Output := FALSE;
            payload.T1_ElapsedTime := T#2s;

            // Apply mock with payload
            AxUnit.Mocking.Mock(
                mockeeFn := NAME_OF(TOF_Mock_true),
                mockFn := NAME_OF(IdentifierBasedTOFMock),
                payload := payload
            );

            // Execute function block in mode 2
            testInstance(mode := 2);

            // Verify result
            Equal(expected := 'MODE2_OFF', actual := testInstance.result);
        END_METHOD

        /// Test Mode 3 - Timer at position 1 should be ON
        {Test}
        METHOD PUBLIC TestMode3TimerOn
            // Reset counter before test
            payload.ResetCounter();

            // Configure Timer 1 (1st call position) to be ON
            payload.T1_Enabled := TRUE;
            payload.T1_CallPosition := 1;
            payload.T1_Output := TRUE;
            payload.T1_ElapsedTime := T#0ms;

            // Apply mock with payload
            AxUnit.Mocking.Mock(
                mockeeFn := NAME_OF(TOF_Mock_true),
                mockFn := NAME_OF(IdentifierBasedTOFMock),
                payload := payload
            );

            // Execute function block in mode 3
            testInstance(mode := 3);

            // Verify result
            Equal(expected := 'MODE3_ON', actual := testInstance.result);
        END_METHOD

        /// Test with multiple configured timers - only matching position is used
        {Test}
        METHOD PUBLIC TestMultipleConfiguredTimers
            // Reset counter before test
            payload.ResetCounter();

            // Configure multiple timers with different call positions
            payload.T1_Enabled := TRUE;
            payload.T1_CallPosition := 1;
            payload.T1_Output := FALSE;
            payload.T1_ElapsedTime := T#1s;

            payload.T2_Enabled := TRUE;
            payload.T2_CallPosition := 2;
            payload.T2_Output := TRUE;
            payload.T2_ElapsedTime := T#0ms;

            // Apply mock with payload
            AxUnit.Mocking.Mock(
                mockeeFn := NAME_OF(TOF_Mock_true),
                mockFn := NAME_OF(IdentifierBasedTOFMock),
                payload := payload
            );

            // Execute function block in mode 2 (should match T1 at position 1, but T1 is at position 1)
            // Since mode 2 calls timer2, it's the 1st call, so T1 matches
            testInstance(mode := 2);

            // Verify result - T1 configuration is used (position 1, OFF)
            Equal(expected := 'MODE2_OFF', actual := testInstance.result);
        END_METHOD
    END_CLASS
END_NAMESPACE

(* ---- IdentifierBasedTONMockTest.st ---- *)
USING AxUnit.Assert;

NAMESPACE Simatic.Ax.Mocks
    /// Example function block with conditional TON timer usage
    FUNCTION_BLOCK ConditionalTONFunctionBlock
        VAR_INPUT
            mode : INT;  // 1, 2, or 3 to select which timer to use
        END_VAR
        VAR_OUTPUT
            result : STRING;
        END_VAR
        VAR
            timer1 : TON_Mock_true;
            timer2 : TON_Mock_true;
            timer3 : TON_Mock_true;
        END_VAR

        // Conditional timer usage based on mode
        IF mode = 1 THEN
            timer1(IN := TRUE, PT := T#1s);
            IF timer1.Q THEN
                result := 'MODE1_ELAPSED';
            ELSE
                result := 'MODE1_WAITING';
            END_IF;
        ELSIF mode = 2 THEN
            timer2(IN := TRUE, PT := T#2s);
            IF timer2.Q THEN
                result := 'MODE2_ELAPSED';
            ELSE
                result := 'MODE2_WAITING';
            END_IF;
        ELSIF mode = 3 THEN
            timer3(IN := TRUE, PT := T#5s);
            IF timer3.Q THEN
                result := 'MODE3_ELAPSED';
            ELSE
                result := 'MODE3_WAITING';
            END_IF;
        ELSE
            result := 'INVALID_MODE';
        END_IF;
    END_FUNCTION_BLOCK

    /// Test fixture demonstrating IdentifierBasedTONMock usage
    {TestFixture}
    CLASS TestIdentifierBasedTONMock
        VAR
            testInstance, testInstanceStateless : ConditionalTONFunctionBlock;
            payload, payloadStateless : IdentifierBasedTONMockPayload;
        END_VAR

        /// Setup method to reset instances before each test
        {TestSetup}
        METHOD PUBLIC TestSetup
            payload := payloadStateless;
            testInstance := testInstanceStateless;
        END_METHOD

        /// Test Mode 1 - Timer at position 1 should be elapsed
        {Test}
        METHOD PUBLIC TestMode1TimerElapsed
            // Reset counter before test
            payload.ResetCounter();

            // Configure Timer 1 (1st call position) to be elapsed
            payload.T1_Enabled := TRUE;
            payload.T1_CallPosition := 1;
            payload.T1_Output := TRUE;
            payload.T1_ElapsedTime := T#1s;

            // Apply mock with payload
            AxUnit.Mocking.Mock(
                mockeeFn := NAME_OF(TON_Mock_true),
                mockFn := NAME_OF(IdentifierBasedTONMock),
                payload := payload
            );

            // Execute function block in mode 1
            testInstance(mode := 1);

            // Verify result
            Equal(expected := 'MODE1_ELAPSED', actual := testInstance.result);
        END_METHOD

        /// Test Mode 2 - Timer at position 1 should be waiting
        {Test}
        METHOD PUBLIC TestMode2TimerWaiting
            // Reset counter before test
            payload.ResetCounter();

            // Configure Timer 1 (1st call position) to be waiting
            payload.T1_Enabled := TRUE;
            payload.T1_CallPosition := 1;
            payload.T1_Output := FALSE;
            payload.T1_ElapsedTime := T#1s;

            // Apply mock with payload
            AxUnit.Mocking.Mock(
                mockeeFn := NAME_OF(TON_Mock_true),
                mockFn := NAME_OF(IdentifierBasedTONMock),
                payload := payload
            );

            // Execute function block in mode 2
            testInstance(mode := 2);

            // Verify result
            Equal(expected := 'MODE2_WAITING', actual := testInstance.result);
        END_METHOD

        /// Test Mode 3 - Timer at position 1 should be elapsed
        {Test}
        METHOD PUBLIC TestMode3TimerElapsed
            // Reset counter before test
            payload.ResetCounter();

            // Configure Timer 1 (1st call position) to be elapsed
            payload.T1_Enabled := TRUE;
            payload.T1_CallPosition := 1;
            payload.T1_Output := TRUE;
            payload.T1_ElapsedTime := T#5s;

            // Apply mock with payload
            AxUnit.Mocking.Mock(
                mockeeFn := NAME_OF(TON_Mock_true),
                mockFn := NAME_OF(IdentifierBasedTONMock),
                payload := payload
            );

            // Execute function block in mode 3
            testInstance(mode := 3);

            // Verify result
            Equal(expected := 'MODE3_ELAPSED', actual := testInstance.result);
        END_METHOD

        /// Test with multiple configured timers - only matching position is used
        {Test}
        METHOD PUBLIC TestMultipleConfiguredTimers
            // Reset counter before test
            payload.ResetCounter();

            // Configure multiple timers with different call positions
            payload.T1_Enabled := TRUE;
            payload.T1_CallPosition := 1;
            payload.T1_Output := FALSE;
            payload.T1_ElapsedTime := T#500ms;

            payload.T2_Enabled := TRUE;
            payload.T2_CallPosition := 2;
            payload.T2_Output := TRUE;
            payload.T2_ElapsedTime := T#2s;

            // Apply mock with payload
            AxUnit.Mocking.Mock(
                mockeeFn := NAME_OF(TON_Mock_true),
                mockFn := NAME_OF(IdentifierBasedTONMock),
                payload := payload
            );

            // Execute function block in mode 2 (should match T1 at position 1)
            // Since mode 2 calls timer2, it's the 1st call, so T1 matches
            testInstance(mode := 2);

            // Verify result - T1 configuration is used (position 1, waiting)
            Equal(expected := 'MODE2_WAITING', actual := testInstance.result);
        END_METHOD
    END_CLASS
END_NAMESPACE

(* ---- IEC_TON_Mocks_Test.st ---- *)
USING AxUnit.Assert;

NAMESPACE Simatic.Ax.Mocks.Tests
    /// Test fixture for IEC TON (On-Delay Timer) Mocks
    /// Tests both TON_Mock_false and TON_Mock_true
    {TestFixture}
    CLASS TestIEC_TON_Mocks
        VAR
            ton_false, ton_false_stateless : TON_Mock_false;
            ton_true, ton_true_stateless : TON_Mock_true;
        END_VAR

        {TestSetup}
        METHOD PUBLIC TestSetup
            ton_false := ton_false_stateless;
            ton_true := ton_true_stateless;
        END_METHOD

        /// Test TON_Mock_false always returns Q=FALSE
        {Test}
        METHOD PUBLIC Test_TON_False_ReturnsAlwaysFalse
            // Call with IN=TRUE
            ton_false(IN := TRUE, PT := T#5s);

            // Verify output is always FALSE
            Equal(expected := FALSE, actual := ton_false.Q);
            Equal(expected := T#0ms, actual := ton_false.ET);
        END_METHOD

        /// Test TON_Mock_false with IN=FALSE
        {Test}
        METHOD PUBLIC Test_TON_False_WithInputFalse
            // Call with IN=FALSE
            ton_false(IN := FALSE, PT := T#10s);

            // Verify output is FALSE
            Equal(expected := FALSE, actual := ton_false.Q);
            Equal(expected := T#0ms, actual := ton_false.ET);
        END_METHOD

        /// Test TON_Mock_true always returns Q=TRUE
        {Test}
        METHOD PUBLIC Test_TON_True_ReturnsAlwaysTrue
            // Call with IN=TRUE
            ton_true(IN := TRUE, PT := T#5s);

            // Verify output is always TRUE and ET equals PT
            Equal(expected := TRUE, actual := ton_true.Q);
            Equal(expected := T#5s, actual := ton_true.ET);
        END_METHOD

        /// Test TON_Mock_true with IN=FALSE
        {Test}
        METHOD PUBLIC Test_TON_True_WithInputFalse
            // Call with IN=FALSE
            ton_true(IN := FALSE, PT := T#10s);

            // Verify output is still TRUE (mock behavior)
            Equal(expected := TRUE, actual := ton_true.Q);
            Equal(expected := T#10s, actual := ton_true.ET);
        END_METHOD

        /// Test TON_Mock_true with different PT values
        {Test}
        METHOD PUBLIC Test_TON_True_DifferentPresetTimes
            // Test with 1 second
            ton_true(IN := TRUE, PT := T#1s);
            Equal(expected := TRUE, actual := ton_true.Q);
            Equal(expected := T#1s, actual := ton_true.ET);

            // Test with 30 seconds
            ton_true(IN := TRUE, PT := T#30s);
            Equal(expected := TRUE, actual := ton_true.Q);
            Equal(expected := T#30s, actual := ton_true.ET);
        END_METHOD

        /// Test TON_Mock_false with different PT values
        {Test}
        METHOD PUBLIC Test_TON_False_DifferentPresetTimes
            // Test with 1 second
            ton_false(IN := TRUE, PT := T#1s);
            Equal(expected := FALSE, actual := ton_false.Q);
            Equal(expected := T#0ms, actual := ton_false.ET);

            // Test with 30 seconds
            ton_false(IN := TRUE, PT := T#30s);
            Equal(expected := FALSE, actual := ton_false.Q);
            Equal(expected := T#0ms, actual := ton_false.ET);
        END_METHOD
    END_CLASS
END_NAMESPACE

(* ---- OnDelayMockWithTwoTimersTest.st ---- *)
USING System.Timer;
USING Simatic.Ax.Mocks;
NAMESPACE Simatic.Ax.Example
    /// Test fixture for testing OnDelayMock with two timers and verifying their states.
    {TestFixture}
    CLASS TestActiveWait
        VAR
            _payloadinstance : OnDelayMockState;
            testInstance : Testee;
        END_VAR

        /// Tests the state of two timers after one clock cycle with mocked values.
        /// Input: None.
        /// Returns: None. Asserts expected timer states.
        {Test}
        METHOD PUBLIC Test_One_Clock_Cycle_Expect_True_False_True
            // give the timer instances a uniq ID. For this purpose, the duration will be used.
            // This is possible, because the result of the timer depends on the mock and not on the time
            testInstance.ValueT1 := T#1s;
            testInstance.ValueT2 := T#2s;

            // Mock timer values after 5 seconds: Timer1 returns true, Timer2 returns false
            _payloadinstance.StatusTimer1 := TRUE;
            _payloadinstance.StatusTimer2 := FALSE;

            // Mock-Setup
            AxUnit.Mocking.Mock(NAME_OF(OnDelay), NAME_OF(OnDelayMock2Timer), _payloadinstance);
            testInstance.Execute(run := TRUE);
            AxUnit.Assert.Equal(expected := TRUE, actual := testInstance.GetTimerState(1));  // expected true --> but something went wrong
            // AxUnit.Assert.Equal(expected := FALSE, actual := testInstance.GetTimerState(2));

        END_METHOD
    END_CLASS

    /// Class under test that manages two OnDelay timers and exposes their states.
    CLASS Testee
      VAR PUBLIC
        /// Duration for timer 1.
        ValueT1 : LTIME := T#1s;
        /// Duration for timer 2.
        ValueT2 : LTIME := T#2s;
      END_VAR

      VAR
        t1 : Ondelay;
        t2 : OnDelay;
      END_VAR

      /// Executes both timers with the provided run signal and configured durations.
      /// Input: run - BOOL signal to start both timers.
      /// Returns: None.
      METHOD PUBLIC Execute
        VAR_INPUT
          run : BOOL;
        END_VAR
        t1(signal := run, duration := ValueT1);
        t2(signal := run, duration := ValueT2);
      END_METHOD

      /// Gets the output state of the specified timer.
      /// Input: id - INT, 1 for t1, 2 for t2.
      /// Returns: BOOL state of the selected timer.
      METHOD PUBLIC GetTimerState : BOOL
        VAR_INPUT
          id : INT;
        END_VAR

        CASE id OF
          1 : GetTimerState := t1.output;
          2 : GetTimerState := t2.output;
        END_CASE;
      END_METHOD

    END_CLASS

END_NAMESPACE

(* ---- SimpleMocks_RealWorld_Test.st ---- *)
USING AxUnit.Assert;
USING System.Timer;

NAMESPACE Simatic.Ax.Mocks.Tests
    /// Example function block with a single OnDelay timer
    /// Demonstrates typical single-timer usage
    FUNCTION_BLOCK SingleTimerController
        VAR_INPUT
            enable : BOOL;
        END_VAR
        VAR_OUTPUT
            status : STRING;
            isReady : BOOL;
        END_VAR
        VAR
            startupTimer : OnDelay;
        END_VAR

        // Single timer for startup delay
        startupTimer(signal := enable, duration := T#5s);

        IF startupTimer.output THEN
            status := 'READY';
            isReady := TRUE;
        ELSIF enable AND NOT startupTimer.output THEN
            status := 'STARTING';
            isReady := FALSE;
        ELSE
            status := 'IDLE';
            isReady := FALSE;
        END_IF;
    END_FUNCTION_BLOCK

    /// Example function block with multiple timers that should ALL have the same state
    /// Use case: All timers must be elapsed before proceeding
    FUNCTION_BLOCK MultiTimerAllSameState
        VAR_INPUT
            enable : BOOL;
        END_VAR
        VAR_OUTPUT
            allReady : BOOL;
            status : STRING;
        END_VAR
        VAR
            timer1 : OnDelay;
            timer2 : OnDelay;
            timer3 : OnDelay;
        END_VAR

        // All timers must be elapsed for system to be ready
        timer1(signal := enable, duration := T#5s);
        timer2(signal := enable, duration := T#10s);
        timer3(signal := enable, duration := T#15s);

        // Check if ALL timers are elapsed
        IF timer1.output AND timer2.output AND timer3.output THEN
            allReady := TRUE;
            status := 'ALL_READY';
        ELSE
            allReady := FALSE;
            status := 'WAITING';
        END_IF;
    END_FUNCTION_BLOCK

    /// Test fixture for simple timer mocks with realistic function blocks
    /// Demonstrates when simple mocks should be used
    {TestFixture}
    CLASS TestSimpleMocks_RealWorld
        VAR
            singleTimer, singleTimerStateless : SingleTimerController;
            multiTimerSame, multiTimerSameStateless : MultiTimerAllSameState;
        END_VAR

        {TestSetup}
        METHOD PUBLIC TestSetup
            singleTimer := singleTimerStateless;
            multiTimerSame := multiTimerSameStateless;
        END_METHOD

        /// ✅ CORRECT USAGE: Single timer - test elapsed state
        {Test}
        METHOD PUBLIC Test_SingleTimer_Elapsed
            // Mock single timer as elapsed
            AxUnit.Mocking.Mock(NAME_OF(OnDelay), NAME_OF(OnDelayMock_true));

            singleTimer(enable := TRUE);

            Equal(expected := 'READY', actual := singleTimer.status);
            Equal(expected := TRUE, actual := singleTimer.isReady);
        END_METHOD

        /// ✅ CORRECT USAGE: Single timer - test waiting state
        {Test}
        METHOD PUBLIC Test_SingleTimer_Waiting
            // Mock single timer as not elapsed
            AxUnit.Mocking.Mock(NAME_OF(OnDelay), NAME_OF(OnDelayMock_false));

            singleTimer(enable := TRUE);

            Equal(expected := 'STARTING', actual := singleTimer.status);
            Equal(expected := FALSE, actual := singleTimer.isReady);
        END_METHOD

        /// ✅ CORRECT USAGE: Multiple timers ALL elapsed (same state)
        {Test}
        METHOD PUBLIC Test_MultipleTimers_AllElapsed
            // Mock ALL timers as elapsed
            AxUnit.Mocking.Mock(NAME_OF(OnDelay), NAME_OF(OnDelayMock_true));

            multiTimerSame(enable := TRUE);

            Equal(expected := TRUE, actual := multiTimerSame.allReady);
            Equal(expected := 'ALL_READY', actual := multiTimerSame.status);
        END_METHOD

        /// ✅ CORRECT USAGE: Multiple timers ALL waiting (same state)
        {Test}
        METHOD PUBLIC Test_MultipleTimers_AllWaiting
            // Mock ALL timers as not elapsed
            AxUnit.Mocking.Mock(NAME_OF(OnDelay), NAME_OF(OnDelayMock_false));

            multiTimerSame(enable := TRUE);

            Equal(expected := FALSE, actual := multiTimerSame.allReady);
            Equal(expected := 'WAITING', actual := multiTimerSame.status);
        END_METHOD

        /// ❌ LIMITATION EXAMPLE: Cannot test mixed states with simple mocks
        /// For this scenario, use ConfigurableTimerMock or IdentifierBasedTimerMock
        {Test}
        METHOD PUBLIC Test_Limitation_CannotTestMixedStates
            // Simple mocks set ALL timers to the same state
            // Cannot test: timer1=TRUE, timer2=FALSE, timer3=TRUE

            // This test demonstrates the limitation:
            AxUnit.Mocking.Mock(NAME_OF(OnDelay), NAME_OF(OnDelayMock_true));

            multiTimerSame(enable := TRUE);

            // All timers will be TRUE (cannot have mixed states)
            Equal(expected := TRUE, actual := multiTimerSame.allReady);

            // ⚠️ If you need mixed states, use ConfigurableTimerMock instead!
        END_METHOD
    END_CLASS

    /// Additional example: Emergency stop with single timer
    FUNCTION_BLOCK EmergencyStopController
        VAR_INPUT
            emergencyStop : BOOL;
        END_VAR
        VAR_OUTPUT
            safeToRestart : BOOL;
            message : STRING;
        END_VAR
        VAR
            cooldownTimer : OffDelay;
        END_VAR

        // Off-delay timer for cooldown after emergency stop
        cooldownTimer(signal := NOT emergencyStop, duration := T#30s);

        IF cooldownTimer.output THEN
            safeToRestart := TRUE;
            message := 'SAFE_TO_RESTART';
        ELSE
            safeToRestart := FALSE;
            message := 'COOLDOWN_ACTIVE';
        END_IF;
    END_FUNCTION_BLOCK

    /// Test fixture for OffDelay simple mocks
    {TestFixture}
    CLASS TestSimpleMocks_OffDelay
        VAR
            emergencyStop, emergencyStopStateless : EmergencyStopController;
        END_VAR

        {TestSetup}
        METHOD PUBLIC TestSetup
            emergencyStop := emergencyStopStateless;
        END_METHOD

        /// ✅ CORRECT USAGE: Single OffDelay timer - cooldown complete
        {Test}
        METHOD PUBLIC Test_EmergencyStop_CooldownComplete
            // Mock timer as elapsed (safe to restart)
            AxUnit.Mocking.Mock(NAME_OF(OffDelay), NAME_OF(OffDelayMock_true));

            emergencyStop(emergencyStop := FALSE);

            Equal(expected := TRUE, actual := emergencyStop.safeToRestart);
            Equal(expected := 'SAFE_TO_RESTART', actual := emergencyStop.message);
        END_METHOD

        /// ✅ CORRECT USAGE: Single OffDelay timer - cooldown active
        {Test}
        METHOD PUBLIC Test_EmergencyStop_CooldownActive
            // Mock timer as not elapsed (still cooling down)
            AxUnit.Mocking.Mock(NAME_OF(OffDelay), NAME_OF(OffDelayMock_false));

            emergencyStop(emergencyStop := FALSE);

            Equal(expected := FALSE, actual := emergencyStop.safeToRestart);
            Equal(expected := 'COOLDOWN_ACTIVE', actual := emergencyStop.message);
        END_METHOD
    END_CLASS
END_NAMESPACE

(* ---- System_OffDelay_Mocks_Test.st ---- *)
USING AxUnit.Assert;
USING System.Timer;

NAMESPACE Simatic.Ax.Mocks.Tests
    /// Test fixture for System.Timer OffDelay Mocks
    /// Tests both OffDelayMock_false and OffDelayMock_true
    {TestFixture}
    CLASS TestSystem_OffDelay_Mocks
        VAR
            offdelay_false, offdelay_false_stateless : OffDelayMock_false;
            offdelay_true, offdelay_true_stateless : OffDelayMock_true;
        END_VAR

        {TestSetup}
        METHOD PUBLIC TestSetup
            offdelay_false := offdelay_false_stateless;
            offdelay_true := offdelay_true_stateless;
        END_METHOD

        /// Test OffDelayMock_false always returns output=FALSE
        {Test}
        METHOD PUBLIC Test_OffDelay_False_ReturnsAlwaysFalse
            // Call with signal=TRUE
            offdelay_false(signal := TRUE, duration := T#5s);

            // Verify output is always FALSE
            Equal(expected := FALSE, actual := offdelay_false.output);
            Equal(expected := T#0ms, actual := offdelay_false.elapsedTime);
        END_METHOD

        /// Test OffDelayMock_false with signal=FALSE
        {Test}
        METHOD PUBLIC Test_OffDelay_False_WithSignalFalse
            // Call with signal=FALSE
            offdelay_false(signal := FALSE, duration := T#10s);

            // Verify output is FALSE
            Equal(expected := FALSE, actual := offdelay_false.output);
            Equal(expected := T#0ms, actual := offdelay_false.elapsedTime);
        END_METHOD

        /// Test OffDelayMock_true always returns output=TRUE
        {Test}
        METHOD PUBLIC Test_OffDelay_True_ReturnsAlwaysTrue
            // Call with signal=TRUE
            offdelay_true(signal := TRUE, duration := T#5s);

            // Verify output is always TRUE and elapsedTime equals duration
            Equal(expected := TRUE, actual := offdelay_true.output);
            Equal(expected := T#5s, actual := offdelay_true.elapsedTime);
        END_METHOD

        /// Test OffDelayMock_true with signal=FALSE
        {Test}
        METHOD PUBLIC Test_OffDelay_True_WithSignalFalse
            // Call with signal=FALSE
            offdelay_true(signal := FALSE, duration := T#10s);

            // Verify output is still TRUE (mock behavior)
            Equal(expected := TRUE, actual := offdelay_true.output);
            Equal(expected := T#10s, actual := offdelay_true.elapsedTime);
        END_METHOD

        /// Test OffDelayMock_true with different duration values
        {Test}
        METHOD PUBLIC Test_OffDelay_True_DifferentDurations
            // Test with 1 second
            offdelay_true(signal := TRUE, duration := T#1s);
            Equal(expected := TRUE, actual := offdelay_true.output);
            Equal(expected := T#1s, actual := offdelay_true.elapsedTime);

            // Test with 30 seconds
            offdelay_true(signal := TRUE, duration := T#30s);
            Equal(expected := TRUE, actual := offdelay_true.output);
            Equal(expected := T#30s, actual := offdelay_true.elapsedTime);
        END_METHOD

        /// Test OffDelayMock_false with different duration values
        {Test}
        METHOD PUBLIC Test_OffDelay_False_DifferentDurations
            // Test with 1 second
            offdelay_false(signal := TRUE, duration := T#1s);
            Equal(expected := FALSE, actual := offdelay_false.output);
            Equal(expected := T#0ms, actual := offdelay_false.elapsedTime);

            // Test with 30 seconds
            offdelay_false(signal := TRUE, duration := T#30s);
            Equal(expected := FALSE, actual := offdelay_false.output);
            Equal(expected := T#0ms, actual := offdelay_false.elapsedTime);
        END_METHOD

        /// Test OffDelayMock_true with LTIME values
        {Test}
        METHOD PUBLIC Test_OffDelay_True_WithLTIME
            // Test with milliseconds
            offdelay_true(signal := TRUE, duration := LTIME#500ms);
            Equal(expected := TRUE, actual := offdelay_true.output);
            Equal(expected := LTIME#500ms, actual := offdelay_true.elapsedTime);

            // Test with minutes
            offdelay_true(signal := TRUE, duration := LTIME#2m);
            Equal(expected := TRUE, actual := offdelay_true.output);
            Equal(expected := LTIME#2m, actual := offdelay_true.elapsedTime);
        END_METHOD
    END_CLASS
END_NAMESPACE

(* ---- System_OnDelay_Mocks_Test.st ---- *)
USING AxUnit.Assert;
USING System.Timer;

NAMESPACE Simatic.Ax.Mocks.Tests
    /// Test fixture for System.Timer OnDelay Mocks
    /// Tests both OnDelayMock_false and OnDelayMock_true
    {TestFixture}
    CLASS TestSystem_OnDelay_Mocks
        VAR
            ondelay_false, ondelay_false_stateless : OnDelayMock_false;
            ondelay_true, ondelay_true_stateless : OnDelayMock_true;
        END_VAR

        {TestSetup}
        METHOD PUBLIC TestSetup
            ondelay_false := ondelay_false_stateless;
            ondelay_true := ondelay_true_stateless;
        END_METHOD

        /// Test OnDelayMock_false always returns output=FALSE
        {Test}
        METHOD PUBLIC Test_OnDelay_False_ReturnsAlwaysFalse
            // Call with signal=TRUE
            ondelay_false(signal := TRUE, duration := T#5s);

            // Verify output is always FALSE
            Equal(expected := FALSE, actual := ondelay_false.output);
            Equal(expected := T#0ms, actual := ondelay_false.elapsedTime);
        END_METHOD

        /// Test OnDelayMock_false with signal=FALSE
        {Test}
        METHOD PUBLIC Test_OnDelay_False_WithSignalFalse
            // Call with signal=FALSE
            ondelay_false(signal := FALSE, duration := T#10s);

            // Verify output is FALSE
            Equal(expected := FALSE, actual := ondelay_false.output);
            Equal(expected := T#0ms, actual := ondelay_false.elapsedTime);
        END_METHOD

        /// Test OnDelayMock_true always returns output=TRUE
        {Test}
        METHOD PUBLIC Test_OnDelay_True_ReturnsAlwaysTrue
            // Call with signal=TRUE
            ondelay_true(signal := TRUE, duration := T#5s);

            // Verify output is always TRUE and elapsedTime equals duration
            Equal(expected := TRUE, actual := ondelay_true.output);
            Equal(expected := T#5s, actual := ondelay_true.elapsedTime);
        END_METHOD

        /// Test OnDelayMock_true with signal=FALSE
        {Test}
        METHOD PUBLIC Test_OnDelay_True_WithSignalFalse
            // Call with signal=FALSE
            ondelay_true(signal := FALSE, duration := T#10s);

            // Verify output is still TRUE (mock behavior)
            Equal(expected := TRUE, actual := ondelay_true.output);
            Equal(expected := T#10s, actual := ondelay_true.elapsedTime);
        END_METHOD

        /// Test OnDelayMock_true with different duration values
        {Test}
        METHOD PUBLIC Test_OnDelay_True_DifferentDurations
            // Test with 1 second
            ondelay_true(signal := TRUE, duration := T#1s);
            Equal(expected := TRUE, actual := ondelay_true.output);
            Equal(expected := T#1s, actual := ondelay_true.elapsedTime);

            // Test with 30 seconds
            ondelay_true(signal := TRUE, duration := T#30s);
            Equal(expected := TRUE, actual := ondelay_true.output);
            Equal(expected := T#30s, actual := ondelay_true.elapsedTime);
        END_METHOD

        /// Test OnDelayMock_false with different duration values
        {Test}
        METHOD PUBLIC Test_OnDelay_False_DifferentDurations
            // Test with 1 second
            ondelay_false(signal := TRUE, duration := T#1s);
            Equal(expected := FALSE, actual := ondelay_false.output);
            Equal(expected := T#0ms, actual := ondelay_false.elapsedTime);

            // Test with 30 seconds
            ondelay_false(signal := TRUE, duration := T#30s);
            Equal(expected := FALSE, actual := ondelay_false.output);
            Equal(expected := T#0ms, actual := ondelay_false.elapsedTime);
        END_METHOD

        /// Test OnDelayMock_true with LTIME values
        {Test}
        METHOD PUBLIC Test_OnDelay_True_WithLTIME
            // Test with milliseconds
            ondelay_true(signal := TRUE, duration := LTIME#500ms);
            Equal(expected := TRUE, actual := ondelay_true.output);
            Equal(expected := LTIME#500ms, actual := ondelay_true.elapsedTime);

            // Test with minutes
            ondelay_true(signal := TRUE, duration := LTIME#2m);
            Equal(expected := TRUE, actual := ondelay_true.output);
            Equal(expected := LTIME#2m, actual := ondelay_true.elapsedTime);
        END_METHOD
    END_CLASS
END_NAMESPACE
